// TIA Portal V20 export
TYPE "LER_typeCommunicationInspection"
// stored: Access Published
   STRUCT
      InspectionToStack : "LER_typeCommunicationDataI2S";
      StackToInspection : "LER_typeCommunicationDataS2I";
   END_STRUCT;
END_TYPE
